{attribute 'linkalways'} 
{attribute 'no_explicit_call' := 'This FB is a CLASS and must be accessed using methods or properties'}
{attribute 'enable_dynamic_creation'}
FUNCTION_BLOCK _TIMESTRUCT EXTENDS StructuredDatatypeBase
VAR
	localData : TIMESTRUCT;
	activeData : REFERENCE TO TIMESTRUCT REF= localData;
	_wYear : _WORD(localData.wYear);
	_wMonth : _WORD(localData.wMonth);
	_wDayOfWeek : _WORD(localData.wDayOfWeek);
	_wDay : _WORD(localData.wDay);
	_wHour : _WORD(localData.wHour);
	_wMinute : _WORD(localData.wMinute);
	_wSecond : _WORD(localData.wSecond);
	_wMilliseconds : _WORD(localData.wMilliseconds);
END_VAR

PROPERTY PUBLIC Address : PVOID
GET
Address := ADR(activeData);
END_GET
END_PROPERTY

METHOD PUBLIC ClearReference
VAR_INPUT
END_VAR
activeData REF= localData;
SetMemberReference();
END_METHOD

METHOD PUBLIC Clone : I_Datatype
VAR
    pClone : POINTER TO _TIMESTRUCT;
END_VAR
pClone := __NEW(_TIMESTRUCT());
pClone^.Value := Value;
Clone := pClone^;
END_METHOD

METHOD FB_init : BOOL
VAR_INPUT
	bInitRetains : BOOL; // if TRUE, the retain variables are initialized (warm start / cold start)
	bInCopyCode : BOOL;  // if TRUE, the instance afterwards gets moved into the copy code (online change)
END_VAR
SetMemberReference();
AddMember('wYear',_wYear);
AddMember('wMonth',_wMonth);
AddMember('wDayOfWeek',_wDayOfWeek);
AddMember('wDay',_wDay);
AddMember('wHour',_wHour);
AddMember('wMinute',_wMinute);
AddMember('wSecond',_wSecond);
AddMember('wMilliseconds',_wMilliseconds);
END_METHOD

PROPERTY PUBLIC Identifier : T_MAXSTRING
GET
Identifier := 'TIMESTRUCT';
END_GET
END_PROPERTY

METHOD PUBLIC MakeReferenceTo
VAR_INPUT
	ReferenceTarget : REFERENCE TO TIMESTRUCT;
END_VAR
activeData REF= ReferenceTarget;
SetMemberReference();
END_METHOD

METHOD PROTECTED SetMemberReference
VAR_INPUT
END_VAR
_wYear.MakeReferenceTo(activeData.wYear);
_wMonth.MakeReferenceTo(activeData.wMonth);
_wDayOfWeek.MakeReferenceTo(activeData.wDayOfWeek);
_wDay.MakeReferenceTo(activeData.wDay);
_wHour.MakeReferenceTo(activeData.wHour);
_wMinute.MakeReferenceTo(activeData.wMinute);
_wSecond.MakeReferenceTo(activeData.wSecond);
_wMilliseconds.MakeReferenceTo(activeData.wMilliseconds);
END_METHOD

PROPERTY PUBLIC Size : UDINT
GET
Size := SIZEOF(activeData);
END_GET
END_PROPERTY

METHOD TryMakeReferenceTo : BOOL
VAR_INPUT
	Target : I_Datatype;
END_VAR
VAR
	pTargetData : POINTER TO TIMESTRUCT;
END_VAR
IF NOT (Target.Datatype = Datatype) THEN
	RETURN;
END_IF

pTargetData := Target.Address;
activeData REF= pTargetData^;
SetMemberReference();
TryMakeReferenceTo := TRUE;
END_METHOD

PROPERTY PUBLIC Value : TIMESTRUCT
GET
Value := activeData;
END_GET
SET
activeData := Value;
END_SET
END_PROPERTY

PROPERTY PUBLIC wDay : Reference to _WORD
GET
wDay REF= _wDay;
END_GET
END_PROPERTY

PROPERTY PUBLIC wDayOfWeek : Reference to _WORD
GET
wDayOfWeek REF= _wDayOfWeek;
END_GET
END_PROPERTY

PROPERTY PUBLIC wHour : Reference to _WORD
GET
wHour REF= _wHour;
END_GET
END_PROPERTY

PROPERTY PUBLIC wMilliseconds : Reference to _WORD
GET
wMilliseconds REF= _wMilliseconds;
END_GET
END_PROPERTY

PROPERTY PUBLIC wMinute : Reference to _WORD
GET
wMinute REF= _wMinute;
END_GET
END_PROPERTY

PROPERTY PUBLIC wMonth : Reference to _WORD
GET
wMonth REF= _wMonth;
END_GET
END_PROPERTY

PROPERTY PUBLIC wSecond : Reference to _WORD
GET
wSecond REF= _wSecond;
END_GET
END_PROPERTY

PROPERTY PUBLIC wYear : Reference to _WORD
GET
wYear REF= _wYear;
END_GET
END_PROPERTY

END_FUNCTION_BLOCK

(* stored: Version 1.1.0.1, ProductVersion 3.1.4024.12
   POU _TIMESTRUCT: Id {82e9ef09-f63f-071f-12cd-f370d2802325}, SpecialFunc None
   Folder Constructor: Id {395e0979-9095-01c3-124d-3ef7fef83c0a}
   Folder Protected: Id {96dedba4-1ea5-0302-010c-f290c7448a78}
   Property Address: Id {b5129746-2857-0022-1d98-5cd0054c1e32}
   Get Get: Id {b9ad7187-0100-02be-2dd1-43dd70cfdd46}
   Method ClearReference: Id {16c22b7d-2069-0e94-0823-7f69befe1715}
   Method Clone: Id {f9cc5498-2141-4519-8b72-11d757b9f1bd}
   Method FB_init: Id {fa2f12a5-8248-079c-058a-ff5fd8f67242}
   Property Identifier: Id {11804f6c-c92e-0f5b-382d-3367d277dbcc}
   Get Get: Id {7977c071-5d37-04dd-33f0-5d682f8e3abf}
   Method MakeReferenceTo: Id {7e8e9cd2-b76b-014b-0b95-9790b062a9ee}
   Method SetMemberReference: Id {a6781b2b-964d-0db3-1dd1-b3def3fb90d7}
   Property Size: Id {3db85a58-3871-08be-0a1b-c8cbab28906e}
   Get Get: Id {c45ad51d-3dc4-00ea-11f7-a16d1bad1963}
   Method TryMakeReferenceTo: Id {8b5d5a6b-3b1b-05bb-2e0f-edb7929e5540}
   Property Value: Id {b58f9a32-1b3b-0a05-0577-0e7b74707ce6}
   Get Get: Id {d1a2ef74-1fb0-0703-20c2-eb9eec1cc598}
   Set Set: Id {4bd1c6bf-61b3-0a38-37ec-840667c35baf}
   Property wDay: Id {e2ffb82e-f057-013a-25ab-1aaabaa2f213}
   Get Get: Id {0a6ed9b0-5bb2-0be8-396b-a001d7051121}
   Property wDayOfWeek: Id {303525a5-b551-0d49-2de8-be51c3f38f26}
   Get Get: Id {b0875f7c-9d2a-01f7-0872-c559a2b228ab}
   Property wHour: Id {442f0489-3b2f-0974-0d75-2f99437990f6}
   Get Get: Id {624d62b9-76fa-059b-2de2-0e7055b2f49c}
   Property wMilliseconds: Id {f2eb5bc4-a63c-0e7a-0e90-1026aa40013c}
   Get Get: Id {fb3ca918-14d6-0a66-0a0a-dacd7799f4ab}
   Property wMinute: Id {2c0e1d05-f680-033b-2336-d846ffa5ca4d}
   Get Get: Id {8928fffd-3ded-0f7d-28ba-f1dcc48f3c37}
   Property wMonth: Id {54bb8911-1454-0b68-0e6e-66985ac5d437}
   Get Get: Id {8a1a1f3d-9a7a-02bf-2086-eb0b47f7f038}
   Property wSecond: Id {e9291c10-fbca-06c8-0e67-f2943469e6fc}
   Get Get: Id {d0aabd22-aa67-029c-2d66-e4bb3858432f}
   Property wYear: Id {3419be73-53a1-06fe-0591-dafdced19fef}
   Get Get: Id {aaabb8ed-77b5-04e0-2779-9412c3abbc56} *)
